Yaskawa INFORM job: kufsa_new2.JBI

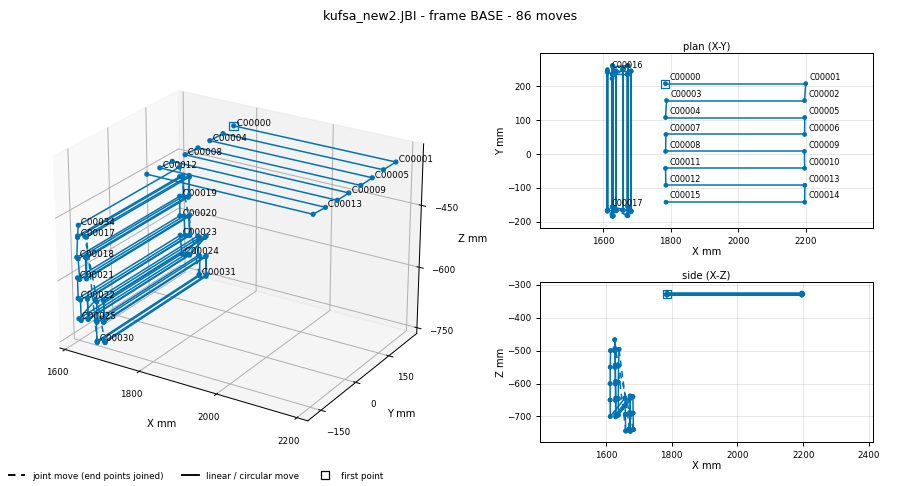
[picture p0: tool path of kufsa_new2.JBI in frame BASE, 86 of 92 moves have a stored position in this frame; points joined in program order, loops and branches not executed]
/JOB
//NAME kufsa_new2
//POS
///NPOS 86,0,86,0,0,0
///TOOL 0
///POSTYPE BASE
///RECTAN
///RCONF 0,0,0,0,0,0,0,0,0,0,0,0,0,0,0,0,0,0,0,0,0,0,0,0
C00000=1784.809984,207.786425,-327.954643,175.000000,5.000000,90.000000
C00001=2198.913977,207.786425,-327.954643,175.000000,5.000000,90.000000
C00002=2195.345305,157.786425,-329.686698,175.000000,5.000000,90.000000
C00003=1788.121031,157.786425,-329.686698,175.000000,5.000000,90.000000
C00004=1785.166089,107.786425,-330.708298,175.000000,5.000000,90.000000
C00005=2195.879591,107.786425,-330.708298,175.000000,5.000000,90.000000
C00006=2195.649886,57.786425,-330.992241,175.000000,5.000000,90.000000
C00007=1786.259788,57.786425,-330.992241,175.000000,5.000000,90.000000
C00008=1785.279038,7.786425,-330.553613,175.000000,5.000000,90.000000
C00009=2194.962549,7.786425,-330.553613,175.000000,5.000000,90.000000
C00010=2195.641002,-42.213575,-329.304422,175.000000,5.000000,90.000000
C00011=1784.984356,-42.213575,-329.304422,175.000000,5.000000,90.000000
C00012=1786.162830,-92.213575,-327.126248,175.000000,5.000000,90.000000
C00013=2196.174273,-92.213575,-327.126248,175.000000,5.000000,90.000000
C00014=2195.835934,-142.213575,-324.584745,175.000000,5.000000,90.000000
C00015=1786.496854,-142.213575,-324.584745,175.000000,5.000000,90.000000
C00016=1614.510230,241.585081,-499.986049,175.000000,-89.999999,5.000000
C00017=1614.510230,-164.000848,-499.986049,175.000000,-89.999999,5.000000
C00018=1613.510109,-168.240064,-549.986049,175.000000,-89.999999,5.000000
C00019=1613.510109,242.364037,-549.986049,175.000000,-89.999999,5.000000
C00020=1613.081853,242.754595,-599.986049,175.000000,-89.999999,5.000000
C00021=1613.081853,-167.653026,-599.986049,175.000000,-89.999999,5.000000
C00022=1613.185617,-167.768560,-649.986049,175.000000,-89.999999,5.000000
C00023=1613.185617,242.941227,-649.986049,175.000000,-89.999999,5.000000
C00024=1613.592087,249.169266,-699.986049,175.000000,-89.999999,5.000000
C00025=1613.592087,-167.776246,-699.986049,175.000000,-89.999999,5.000000
C00026=1658.174221,-165.117278,-643.920031,180.000000,-45.000000,0.000000
C00027=1658.174221,249.874961,-643.920031,180.000000,-45.000000,0.000000
C00028=1659.202806,251.360332,-693.920031,180.000000,-45.000000,0.000000
C00029=1659.202806,-165.909444,-693.920031,180.000000,-45.000000,0.000000
C00030=1660.619905,-166.059086,-743.920031,180.000000,-45.000000,0.000000
C00031=1660.619905,251.190994,-743.920031,180.000000,-45.000000,0.000000
C00032=1660.619905,251.190994,-743.920031,180.000000,-45.000000,0.000000
C00033=1627.039345,222.823878,-466.652847,175.000000,-89.999999,5.000000
C00034=1627.039345,-177.170536,-466.652847,175.000000,-89.999999,5.000000
C00035=1627.487176,-181.874279,-493.857188,175.000000,-89.999999,5.000000
C00036=1627.487176,236.163630,-493.857188,175.000000,-89.999999,5.000000
C00037=1628.694504,234.314063,-543.857188,175.000000,-89.999999,5.000000
C00038=1628.694504,-183.905326,-543.857188,175.000000,-89.999999,5.000000
C00039=1629.893530,-182.345110,-593.857188,175.000000,-89.999999,5.000000
C00040=1629.893530,235.364359,-593.857188,175.000000,-89.999999,5.000000
C00041=1630.508634,236.780914,-643.857188,175.000000,-89.999999,5.000000
C00042=1630.508634,-182.673804,-643.857188,175.000000,-89.999999,5.000000
C00043=1630.668453,-182.518468,-693.857188,175.000000,-89.999999,5.000000
C00044=1630.668453,235.781635,-693.857188,175.000000,-89.999999,5.000000
C00045=1674.177866,234.266599,-637.791171,180.000000,-45.000000,0.000000
C00046=1674.177866,-182.039007,-637.791171,180.000000,-45.000000,0.000000
C00047=1672.996282,-181.752954,-687.791171,180.000000,-45.000000,0.000000
C00048=1672.996282,235.770467,-687.791171,180.000000,-45.000000,0.000000
C00049=1671.625118,235.650157,-737.791171,180.000000,-45.000000,0.000000
C00050=1671.625118,-180.962313,-737.791171,180.000000,-45.000000,0.000000
C00051=1671.625118,-180.962313,-737.791171,180.000000,-45.000000,0.000000
C00052=1640.115541,-166.670113,-496.018038,175.000000,-89.999999,5.000000
C00053=1640.115541,243.723336,-496.018038,175.000000,-89.999999,5.000000
C00054=1638.720755,240.285413,-546.018038,175.000000,-89.999999,5.000000
C00055=1638.720755,-166.379476,-546.018038,175.000000,-89.999999,5.000000
C00056=1638.145643,-168.031063,-596.018038,175.000000,-89.999999,5.000000
C00057=1638.145643,243.325091,-596.018038,175.000000,-89.999999,5.000000
C00058=1638.045149,245.954996,-646.018038,175.000000,-89.999999,5.000000
C00059=1638.045149,-166.457540,-646.018038,175.000000,-89.999999,5.000000
C00060=1638.070457,-166.215422,-696.018038,175.000000,-89.999999,5.000000
C00061=1638.070457,244.005086,-696.018038,175.000000,-89.999999,5.000000
C00062=1682.397576,243.743993,-639.952020,180.000000,-45.000000,0.000000
C00063=1682.397576,-166.492608,-639.952020,180.000000,-45.000000,0.000000
C00064=1682.992057,-170.636948,-689.952020,180.000000,-45.000000,0.000000
C00065=1682.992057,245.671564,-689.952020,180.000000,-45.000000,0.000000
C00066=1683.918555,244.606296,-739.952020,180.000000,-45.000000,0.000000
C00067=1683.918555,-168.420661,-739.952020,180.000000,-45.000000,0.000000
C00068=1683.918555,-168.420661,-739.952020,180.000000,-45.000000,0.000000
C00069=1628.131473,-156.288290,-500.819781,175.000000,-89.999999,5.000000
C00070=1628.131473,261.241476,-500.819781,175.000000,-89.999999,5.000000
C00071=1628.284561,260.410224,-550.819781,175.000000,-89.999999,5.000000
C00072=1628.284561,-156.519518,-550.819781,175.000000,-89.999999,5.000000
C00073=1628.912084,-156.474085,-600.819781,175.000000,-89.999999,5.000000
C00074=1628.912084,260.360222,-600.819781,175.000000,-89.999999,5.000000
C00075=1629.713460,257.495132,-650.819781,175.000000,-89.999999,5.000000
C00076=1629.713460,-155.876345,-650.819781,175.000000,-89.999999,5.000000
C00077=1630.275402,-156.095643,-700.819781,175.000000,-89.999999,5.000000
C00078=1630.275402,257.506046,-700.819781,175.000000,-89.999999,5.000000
C00079=1674.450694,261.075987,-644.753764,180.000000,-45.000000,0.000000
C00080=1674.450694,-156.209353,-644.753764,180.000000,-45.000000,0.000000
C00081=1674.460041,-155.949698,-694.753764,180.000000,-45.000000,0.000000
C00082=1674.460041,260.505660,-694.753764,180.000000,-45.000000,0.000000
C00083=1674.382497,261.189444,-744.753764,180.000000,-45.000000,0.000000
C00084=1674.382497,-155.897919,-744.753764,180.000000,-45.000000,0.000000
C00085=1674.382497,-155.897919,-744.753764,180.000000,-45.000000,0.000000
///POSTYPE PULSE
///PULSE
EC00000=0
EC00001=0
EC00002=0
EC00003=0
EC00004=0
EC00005=0
EC00006=0
EC00007=0
EC00008=0
EC00009=0
EC00010=0
EC00011=0
EC00012=0
EC00013=0
EC00014=0
EC00015=0
EC00016=0
EC00017=0
EC00018=0
EC00019=0
EC00020=0
EC00021=0
EC00022=0
EC00023=0
EC00024=0
EC00025=0
EC00026=0
EC00027=0
EC00028=0
EC00029=0
EC00030=0
EC00031=0
EC00032=92160
EC00033=92160
EC00034=92160
EC00035=92160
EC00036=92160
EC00037=92160
EC00038=92160
EC00039=92160
EC00040=92160
EC00041=92160
EC00042=92160
EC00043=92160
EC00044=92160
EC00045=92160
EC00046=92160
EC00047=92160
EC00048=92160
EC00049=92160
EC00050=92160
EC00051=184320
EC00052=184320
EC00053=184320
EC00054=184320
EC00055=184320
EC00056=184320
EC00057=184320
EC00058=184320
EC00059=184320
EC00060=184320
EC00061=184320
EC00062=184320
EC00063=184320
EC00064=184320
EC00065=184320
EC00066=184320
EC00067=184320
EC00068=276480
EC00069=276480
EC00070=276480
EC00071=276480
EC00072=276480
EC00073=276480
EC00074=276480
EC00075=276480
EC00076=276480
EC00077=276480
EC00078=276480
EC00079=276480
EC00080=276480
EC00081=276480
EC00082=276480
EC00083=276480
EC00084=276480
EC00085=368640
//INST
///DATE 2023/01/19 16:31
///ATTR SC,RW,RJ
////FRAME BASE
///GROUP1 RB1,ST1
NOP
MOVJ P009 EX000 VJ=15.00
MOVJ C00000 EC00000 VJ=15.0
CALL JOB:SPYON
MOVL C00001 EC00001 V=150.0
MOVL C00002 EC00002 V=150.0
MOVL C00003 EC00003 V=150.0
MOVL C00004 EC00004 V=150.0
MOVL C00005 EC00005 V=150.0
MOVL C00006 EC00006 V=150.0
MOVL C00007 EC00007 V=150.0
MOVL C00008 EC00008 V=150.0
MOVL C00009 EC00009 V=150.0
MOVL C00010 EC00010 V=150.0
MOVL C00011 EC00011 V=150.0
MOVL C00012 EC00012 V=150.0
MOVL C00013 EC00013 V=150.0
MOVL C00014 EC00014 V=150.0
MOVL C00015 EC00015 V=150.0
CALL JOB:SPYOF
MOVJ P009 VJ=15.00
MOVJ C00016 EC00016 VJ=15.0
CALL JOB:SPYON
MOVL C00017 EC00017 V=150.0
MOVL C00018 EC00018 V=150.0
MOVL C00019 EC00019 V=150.0
MOVL C00020 EC00020 V=150.0
MOVL C00021 EC00021 V=150.0
MOVL C00022 EC00022 V=150.0
MOVL C00023 EC00023 V=150.0
MOVL C00024 EC00024 V=150.0
MOVL C00025 EC00025 V=150.0
MOVL C00026 EC00026 V=150.0
MOVL C00027 EC00027 V=150.0
MOVL C00028 EC00028 V=150.0
MOVL C00029 EC00029 V=150.0
MOVL C00030 EC00030 V=150.0
MOVL C00031 EC00031 V=150.0
CALL JOB:SPYOF
MOVJ P009 VJ=15.00
MOVL C00032 EC00032 V=150.0
MOVJ C00033 EC00033 VJ=15.0
CALL JOB:SPYON
MOVL C00034 EC00034 V=150.0
MOVL C00035 EC00035 V=150.0
MOVL C00036 EC00036 V=150.0
MOVL C00037 EC00037 V=150.0
MOVL C00038 EC00038 V=150.0
MOVL C00039 EC00039 V=150.0
MOVL C00040 EC00040 V=150.0
MOVL C00041 EC00041 V=150.0
MOVL C00042 EC00042 V=150.0
MOVL C00043 EC00043 V=150.0
MOVL C00044 EC00044 V=150.0
MOVL C00045 EC00045 V=150.0
MOVL C00046 EC00046 V=150.0
MOVL C00047 EC00047 V=150.0
MOVL C00048 EC00048 V=150.0
MOVL C00049 EC00049 V=150.0
MOVL C00050 EC00050 V=150.0
CALL JOB:SPYOF
MOVJ P009 VJ=15.00
MOVL C00051 EC00051 V=150.0
MOVJ C00052 EC00052 VJ=15.0
CALL JOB:SPYON
MOVL C00053 EC00053 V=150.0
MOVL C00054 EC00054 V=150.0
MOVL C00055 EC00055 V=150.0
MOVL C00056 EC00056 V=150.0
MOVL C00057 EC00057 V=150.0
MOVL C00058 EC00058 V=150.0
MOVL C00059 EC00059 V=150.0
MOVL C00060 EC00060 V=150.0
MOVL C00061 EC00061 V=150.0
MOVL C00062 EC00062 V=150.0
MOVL C00063 EC00063 V=150.0
MOVL C00064 EC00064 V=150.0
MOVL C00065 EC00065 V=150.0
MOVL C00066 EC00066 V=150.0
MOVL C00067 EC00067 V=150.0
CALL JOB:SPYOF
MOVJ P009 VJ=15.00
MOVL C00068 EC00068 V=150.0
MOVJ C00069 EC00069 VJ=15.0
CALL JOB:SPYON
MOVL C00070 EC00070 V=150.0
MOVL C00071 EC00071 V=150.0
MOVL C00072 EC00072 V=150.0
MOVL C00073 EC00073 V=150.0
MOVL C00074 EC00074 V=150.0
MOVL C00075 EC00075 V=150.0
MOVL C00076 EC00076 V=150.0
MOVL C00077 EC00077 V=150.0
MOVL C00078 EC00078 V=150.0
MOVL C00079 EC00079 V=150.0
MOVL C00080 EC00080 V=150.0
MOVL C00081 EC00081 V=150.0
MOVL C00082 EC00082 V=150.0
MOVL C00083 EC00083 V=150.0
MOVL C00084 EC00084 V=150.0
CALL JOB:SPYOF
MOVJ P009 VJ=15.00
MOVL C00085 EC00085 V=150.0
END
